FUNCTION_BLOCK BoolComparer EXTENDS Object IMPLEMENTS IComparer
VAR
	_ClassName : STRING := __POUNAME();
END_VAR

{attribute 'monitoring' := 'call'}
PROPERTY ClassName : STRING
GET
ClassName := _ClassName;
END_GET
END_PROPERTY

{attribute "object_name" := "Compare"}
METHOD Compare : COMPARISION_RESULT
VAR_INPUT
	left : GENERIC_VALUE;
	right : GENERIC_VALUE;
END_VAR
VAR
	leftPointer : POINTER TO BOOL; 
	rightPointer : POINTER TO BOOL; 
END_VAR
IF left.Address = 0 AND right.Address = 0 THEN
	Compare := COMPARISION_RESULT.EQUALS;
	RETURN;
END_IF

IF left.Address = 0 THEN
	Compare := COMPARISION_RESULT.LEFT_LESS_RIGHT;
	RETURN;	
END_IF

IF right.Address = 0 THEN
	Compare := COMPARISION_RESULT.LEFT_GREATER_RIGHT;
	RETURN;	
END_IF

leftPointer := left.Address;
rightPointer := right.Address;

IF leftPointer^ < rightPointer^ THEN
	Compare := COMPARISION_RESULT.LEFT_LESS_RIGHT;
ELSIF leftPointer^ > rightPointer^ THEN
	Compare := COMPARISION_RESULT.LEFT_GREATER_RIGHT;
ELSE
	Compare := COMPARISION_RESULT.EQUALS;	
END_IF
END_METHOD

{attribute 'monitoring' := 'call'}
PROPERTY Size : ULINT
GET
Size := XSIZEOF(THIS^);
END_GET
END_PROPERTY

END_FUNCTION_BLOCK

(* stored: Version 1.1.0.1
   POU BoolComparer: Id {b24450aa-877e-4dbf-a945-e3d6ba0462d4}, SpecialFunc None
   Property ClassName: Id {4afee12e-0b26-45c8-895f-f54e650a295b}
   Get Get: Id {07ad798a-3c3b-4d44-ba7d-904602efbc06}
   Method Compare: Id {f48eae1f-deb9-4246-bde6-c91900fab6c2}
   Property Size: Id {910da1bd-51d1-4244-858c-df2c2bca4d47}
   Get Get: Id {ece1a941-c310-49ff-ba83-199c5d1387c1} *)
